{attribute 'no_check'}
FUNCTION IO_TO_BP : ST_BeamParams
VAR_INPUT
    IO : ST_BeamParams_IO;
END_VAR
VAR
    idx : UINT;
END_VAR


FOR idx := 1 TO PMPS_GVL.AUX_ATTENUATORS DO
    IO_TO_BP.astAttenuators[idx] := IO_TO_ATT(IO.astAttenuators[idx]);
END_FOR

FOR idx := 1 TO PMPS_GVL.MAX_APERTURES DO
    IO_TO_BP.astApertures[idx] := IO_TO_APT(IO.astApertures[idx]);
END_FOR

IO_TO_BP.aVetoDevices := IO.aVetoDevices;
IO_TO_BP.nTran := IO.nTran;
IO_TO_BP.nCohortInt := ULINT_TO_UDINT(IO.nCohortInt);
IO_TO_BP.neVRange := IO.neVRange;
IO_TO_BP.neV := IO.neV;
IO_TO_BP.nBCRange := IO.nBCRange;
IO_TO_BP.nBeamClass := IO.nBeamClass;
IO_TO_BP.nMachineMode := IO.nMachineMode;
IO_TO_BP.nRate := IO.nRate;
IO_TO_BP.xValid := IO.xValid;
IO_TO_BP.xValidToggle := IO.xValidToggle;

END_FUNCTION

(* stored: Version 1.1.0.1, ProductVersion 3.1.4022.18
   POU IO_TO_BP: Id {9adf1afe-3d64-4ec4-b76c-d1ce92f03d86}, SpecialFunc None *)
